// TIA Portal V17 export
// export: Created 2025-06-26T07:49:18.7274712Z, ExportSetting WithDefaults, DisplayName Totally Integrated Automation Portal, DisplayVersion V17 Update 8, DisplayName TIA Portal Openness, DisplayVersion V17 Update 8, DisplayName TIA Portal Version Control Interface, DisplayVersion V17, DisplayName STEP 7 Professional, DisplayVersion V17 Update 8, DisplayName STEP 7 Safety, DisplayVersion V17 Update 6, DisplayName WinCC Advanced, DisplayVersion V17 Update 8
TYPE "stCalcValue"
// stored: IsFailsafeCompliant false
   STRUCT
      fMin : Real;   // Negative-most value
      fMax : Real;   // Positive-most value
      fValue : Real;   // Actual value
      bError : Bool;   // Value invalid or out of range
      bCheckLimits : Bool := false;   // 1 = set bError if outside min & max, 0 = do nothing
      bLimited : Bool;   // 1 = value is limited, 0 = value is not limited
   END_STRUCT;
END_TYPE
